// TIA Portal V19 export
TYPE "LEXCHANGETRAY_typeConstraintWorkstationIoSignalInterface"
// configuration: LEXCHANGETRAY_typeConstraintWorkstationIoSignalConfigeration
// commands: LEXCHANGETRAY_typeConstraintWorkstationIoSignalManualCommands
// monitoring: LEXCHANGETRAY_typeConstraintWorkstationIoSignalProcessValues
// stored: Access Published
   STRUCT
      configuration : "LEXCHANGETRAY_typeConstraintWorkstationIoSignalConfigeration";
      commands { S7_SetPoint := 'True'} : "LEXCHANGETRAY_typeConstraintWorkstationIoSignalManualCommands";
      monitoring { S7_SetPoint := 'True'} : "LEXCHANGETRAY_typeConstraintWorkstationIoSignalProcessValues";
   END_STRUCT;
END_TYPE
